// TIA Portal V20 export
// export: Created 2025-12-01T14:57:43.5761957Z, ExportSetting None, DisplayName Totally Integrated Automation Portal, DisplayVersion V20 Update 3, DisplayName TIA Portal Openness, DisplayVersion V20 Update 3, DisplayName TIA Portal Version Control Interface, DisplayVersion V20 Update 3, DisplayName STEP 7 Professional, DisplayVersion V20 Update 3, DisplayName STEP 7 Safety, DisplayVersion V20 Update 2, DisplayName WinCC Basic/Comfort/Advanced, DisplayVersion V20 Update 3, DisplayName WinCC Professional, DisplayVersion V20 Update 3, DisplayName WinCC Unified, DisplayVersion V20 Update 3
FUNCTION "FC506_PASAR_ORD_SCR" : Void   // FC506, LAD
{ S7_Optimized_Access := 'FALSE' }
AUTHOR : TLigero
NAME : 20130623
VERSION : 3.1
// stored: AutoNumber false, SetENOAutomatically false
   VAR_INPUT
      NXT_DB_FIFO_Ordenes : UInt;
      NXT_Num_Scanner : UInt;   // Numero de scanner sobre el que se realiza la busqueda
      NXT_Long_FIFO : UInt;
      Datos_Scanner_Cruce : "ROUT_Orden_Fifo_Scanner";
   END_VAR
   VAR_OUTPUT
      Trans_OK : Bool;
   END_VAR
   VAR_TEMP
      Aux_Puntero : DWord;
      N_DB : Word;
      Num_Cola : UDInt;
      Num_Pos_Etiqueta : UInt;
      Num_Pos_Etiqueta_DB : UInt;   // Numero de etiqueta dentro del DB avierto para la busqueda
      Etiqueta_OK : Bool;
      Ordenes : Byte;
      CNT_Fifo : UInt;
      Num_Pos_Etiqueta_FIN : UInt;
      Pos_Ini_Cruce : UInt;
      Aux_contador : UInt;
      retval : Int;
      Datos_NXT_FIFO : "ROUT_Orden_Fifo_Scanner";
      Datos_Pasar_FIFO : "ROUT_Orden_Fifo_Scanner";
   END_VAR
BEGIN

NETWORK
TITLE = Inicializar variables
//==================================================================

      L     uint#1;
      T     #Aux_contador;

      CALL  FILL
      ( BVAL    := #Datos_Scanner_Cruce,
        RET_VAL := #retval,
        BLK     := #Datos_Pasar_FIFO
      );


//==================================================================

NETWORK
TITLE = Casos especiales, la orden que queremos pasar es un vaciado o no hay hueco en la fifo
//==================================================================
// - Si la orden que tenemos que pasar es un vaciado,
//==================================================================

      SET;
      L     #Datos_Scanner_Cruce.Orden;
      L     w#16#FF;
      ==I;
      JC    pasar_orden_vaciar;
//==================================================================

NETWORK
TITLE = Buscamos una posicion de memoria libre en la siguiente fifo
//==================================================================
// sacamos los datos de la posicion de la fifo
saca_datos_nxt_fifo:NOP   0;

      CALL  "FC571_Leer_Datos_Fifo"
      ( DB_FIFO_Ordenes     := #NXT_DB_FIFO_Ordenes,
        Num_Scanner         := #NXT_Num_Scanner,
        Long_FIFO           := #NXT_Long_FIFO,
        Posicion_FIFO       := #Aux_contador,
        Datos_Scanner_Cruce := #Datos_NXT_FIFO
      );

// - Comprobamos si la fifo está ocupada, comprobando el valor de la orden

      SET;
      L     #Datos_NXT_FIFO.Orden;
      L     0;
      ==I;
      JC    Pasar_orden_Fifo;

// - Si tiene orden, tenemos que buscar el siguiente registro
// - Comprobamos si hemos llegado al límite

// - si no hay hueco es un caso especial

      SET;
      L     #Aux_contador;
      L     #NXT_Long_FIFO;
      ==I;
      JC    Sin_hueco_FIFO;

// - incrementamos en uno la posicion para seguir buscando

      SET;
      L     #Aux_contador;
      L     1;
      +I;
      T     #Aux_contador;

      JU    saca_datos_nxt_fifo;

//==================================================================

NETWORK
TITLE = Casos especiales, la orden a pasar es vaciado, o no hay hueco en la siguiente fifo
//==================================================================
// - Para estos dos casos, sacamos los datos de la primera posicion
// - de la fifo, y le cambiamos la orden a vaciado w#16#FF

Sin_hueco_FIFO:NOP   0;
pasar_orden_vaciar:NOP   0;
//==================================================================

      CALL  "FC571_Leer_Datos_Fifo"
      ( DB_FIFO_Ordenes     := #NXT_DB_FIFO_Ordenes,
        Num_Scanner         := #NXT_Num_Scanner,
        Long_FIFO           := #NXT_Long_FIFO,
        Posicion_FIFO       := uint#1,
        Datos_Scanner_Cruce := #Datos_NXT_FIFO
      );

// - Cambiamos la orden
      L     w#16#FF;
      T     #Datos_NXT_FIFO.Orden;

// - volvemos a guardar los datos

      CALL  "FC572_Guardar_Datos_Fifo"
      ( DB_FIFO_Ordenes     := #NXT_DB_FIFO_Ordenes,
        Num_Scanner         := #NXT_Num_Scanner,
        Long_FIFO           := #NXT_Long_FIFO,
        Posicion_FIFO       := uint#1,
        Datos_Scanner_Cruce := #Datos_NXT_FIFO
      );


// seteamos el bit de que hemos hecho el trasvase OK
// y salimos de la función.
      SET;
      S     #Trans_OK;
      BE;

//==================================================================



NETWORK
TITLE = Pasar orden a la siguiente fifo
//==================================================================
// pasamos la orden a la siguiente fifo
Pasar_orden_Fifo:NOP   0;

      CALL  "FC572_Guardar_Datos_Fifo"
      ( DB_FIFO_Ordenes     := #NXT_DB_FIFO_Ordenes,
        Num_Scanner         := #NXT_Num_Scanner,
        Long_FIFO           := #NXT_Long_FIFO,
        Posicion_FIFO       := #Aux_contador,
        Datos_Scanner_Cruce := #Datos_Scanner_Cruce
      );

// seteamos el bit de que hemos hecho el trasvase OK
// y salimos de la función.
      SET;
      S     #Trans_OK;
      BE;

//==================================================================
END_FUNCTION
